// Mitsubishi GX Works2 project: A1-60MR-GX2   PLC: FX3G

PROGRAM MAIN
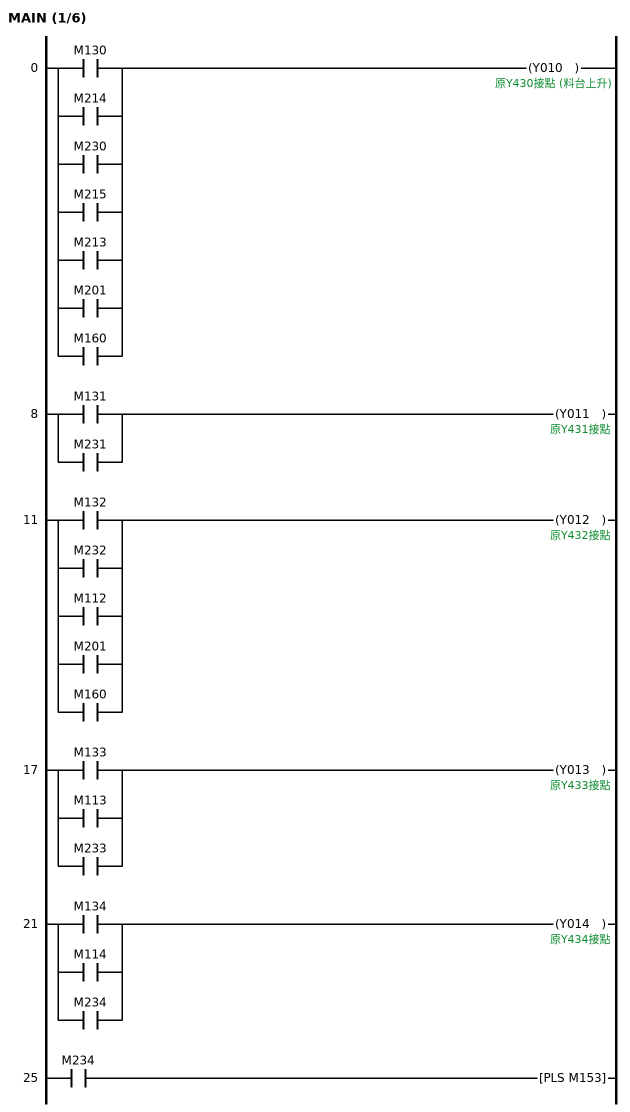
0     LD      M130
      OR      M214
      OR      M230
      OR      M215
      OR      M213
      OR      M201
      OR      M160
      OUT     Y010  ; 原Y430接點 (料台上升)
8     LD      M131
      OR      M231
      OUT     Y011  ; 原Y431接點
11    LD      M132
      OR      M232
      OR      M112
      OR      M201
      OR      M160
      OUT     Y012  ; 原Y432接點
17    LD      M133
      OR      M113
      OR      M233
      OUT     Y013  ; 原Y433接點
21    LD      M134
      OR      M114
      OR      M234
      OUT     Y014  ; 原Y434接點
25    LD      M234
      PLS     M153
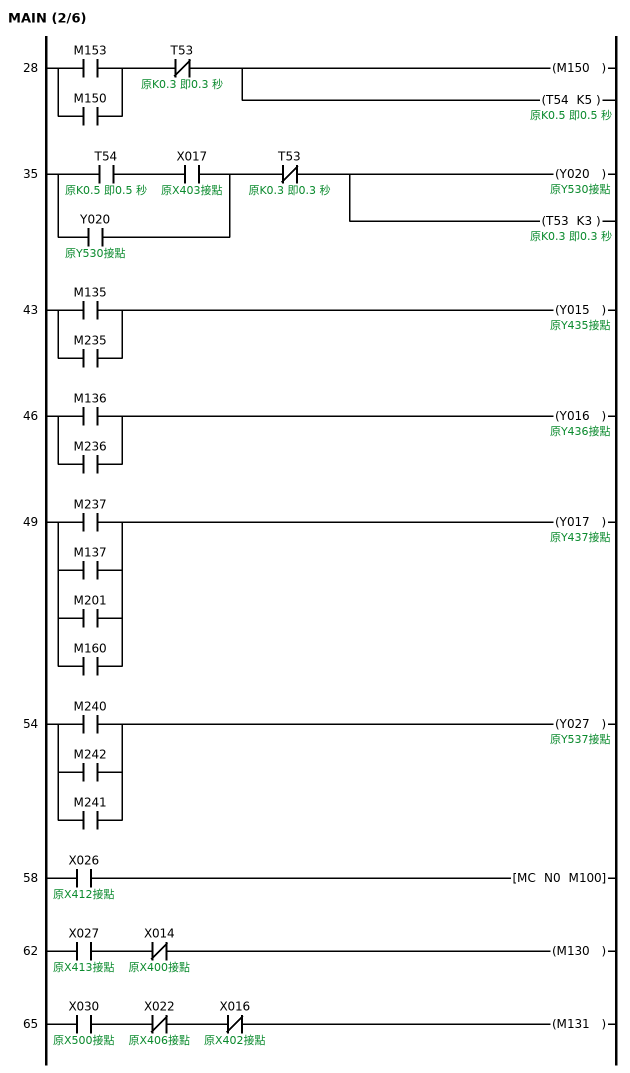
28    LD      M153
      OR      M150
      ANI     T53  ; 原K0.3 即0.3 秒
      OUT     M150
      OUT     T54 K5  ; 原K0.5 即0.5 秒
35    LD      T54  ; 原K0.5 即0.5 秒
      AND     X017  ; 原X403接點
      OR      Y020  ; 原Y530接點
      ANI     T53  ; 原K0.3 即0.3 秒
      OUT     Y020  ; 原Y530接點
      OUT     T53 K3  ; 原K0.3 即0.3 秒
43    LD      M135
      OR      M235
      OUT     Y015  ; 原Y435接點
46    LD      M136
      OR      M236
      OUT     Y016  ; 原Y436接點
49    LD      M237
      OR      M137
      OR      M201
      OR      M160
      OUT     Y017  ; 原Y437接點
54    LD      M240
      OR      M242
      OR      M241
      OUT     Y027  ; 原Y537接點
58    LD      X026  ; 原X412接點
      MC      N0 M100
62    LD      X027  ; 原X413接點
      ANI     X014  ; 原X400接點
      OUT     M130
65    LD      X030  ; 原X500接點
      ANI     X022  ; 原X406接點
      ANI     X016  ; 原X402接點
      OUT     M131
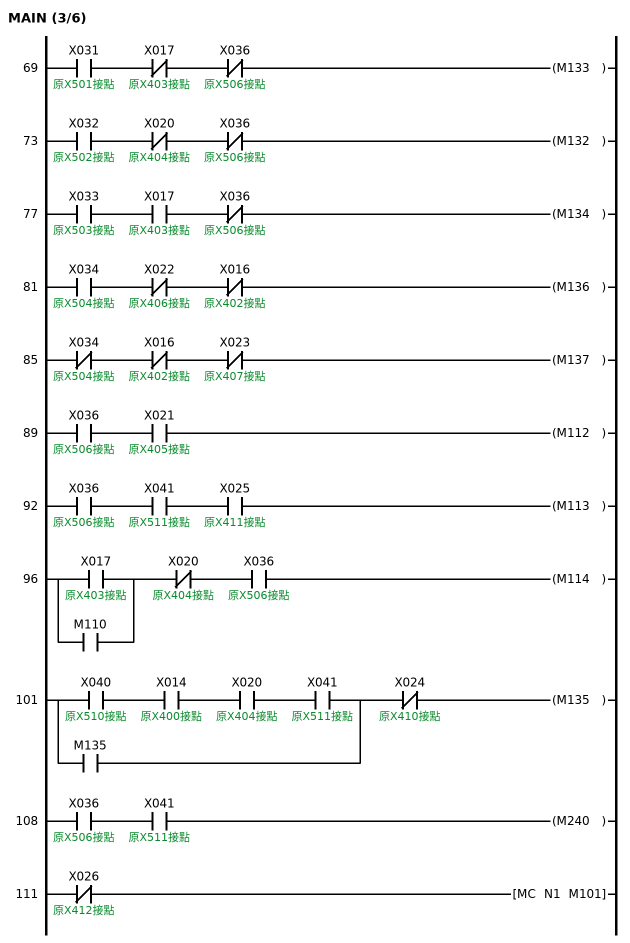
69    LD      X031  ; 原X501接點
      ANI     X017  ; 原X403接點
      ANI     X036  ; 原X506接點
      OUT     M133
73    LD      X032  ; 原X502接點
      ANI     X020  ; 原X404接點
      ANI     X036  ; 原X506接點
      OUT     M132
77    LD      X033  ; 原X503接點
      AND     X017  ; 原X403接點
      ANI     X036  ; 原X506接點
      OUT     M134
81    LD      X034  ; 原X504接點
      ANI     X022  ; 原X406接點
      ANI     X016  ; 原X402接點
      OUT     M136
85    LDI     X034  ; 原X504接點
      ANI     X016  ; 原X402接點
      ANI     X023  ; 原X407接點
      OUT     M137
89    LD      X036  ; 原X506接點
      AND     X021  ; 原X405接點
      OUT     M112
92    LD      X036  ; 原X506接點
      AND     X041  ; 原X511接點
      AND     X025  ; 原X411接點
      OUT     M113
96    LD      X017  ; 原X403接點
      OR      M110
      ANI     X020  ; 原X404接點
      AND     X036  ; 原X506接點
      OUT     M114
101   LD      X040  ; 原X510接點
      AND     X014  ; 原X400接點
      AND     X020  ; 原X404接點
      AND     X041  ; 原X511接點
      OR      M135
      ANI     X024  ; 原X410接點
      OUT     M135
108   LD      X036  ; 原X506接點
      AND     X041  ; 原X511接點
      OUT     M240
111   LDI     X026  ; 原X412接點
      MC      N1 M101
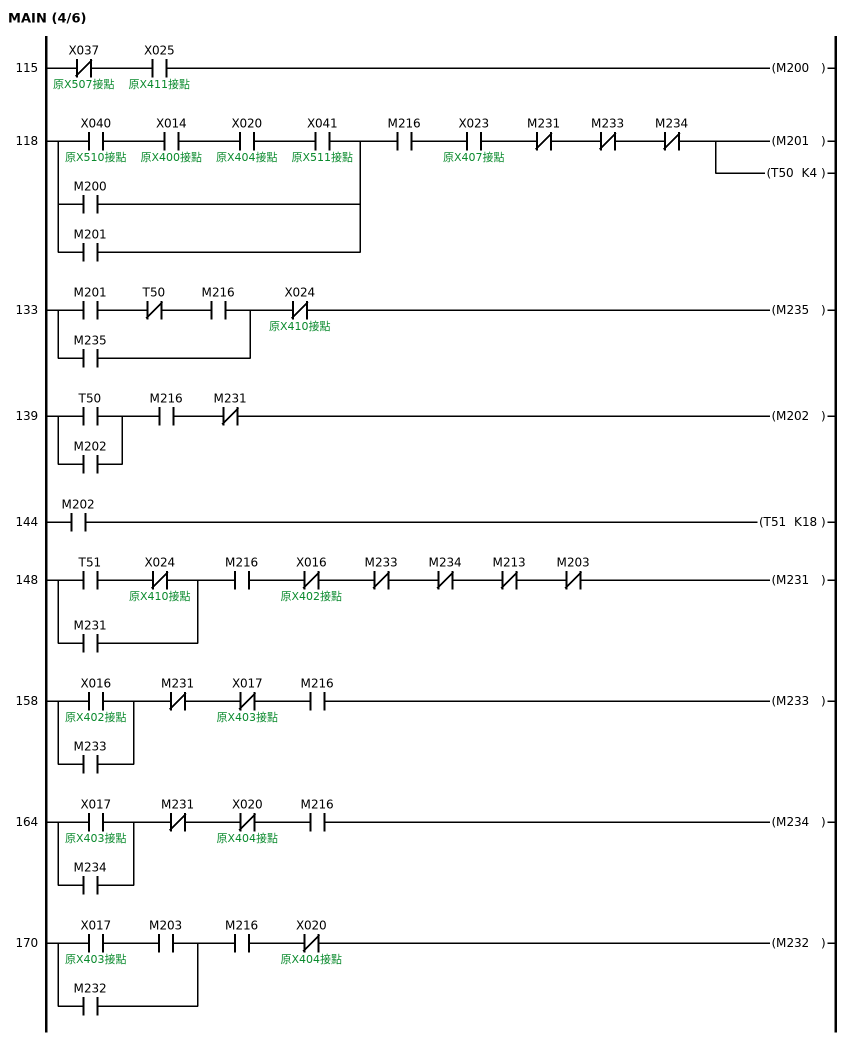
115   LDI     X037  ; 原X507接點
      AND     X025  ; 原X411接點
      OUT     M200
118   LD      X040  ; 原X510接點
      AND     X014  ; 原X400接點
      AND     X020  ; 原X404接點
      AND     X041  ; 原X511接點
      OR      M200
      OR      M201
      AND     M216
      AND     X023  ; 原X407接點
      ANI     M231
      ANI     M233
      ANI     M234
      OUT     M201
      OUT     T50 K4
133   LD      M201
      ANI     T50
      AND     M216
      OR      M235
      ANI     X024  ; 原X410接點
      OUT     M235
139   LD      T50
      OR      M202
      AND     M216
      ANI     M231
      OUT     M202
144   LD      M202
      OUT     T51 K18
148   LD      T51
      ANI     X024  ; 原X410接點
      OR      M231
      AND     M216
      ANI     X016  ; 原X402接點
      ANI     M233
      ANI     M234
      ANI     M213
      ANI     M203
      OUT     M231
158   LD      X016  ; 原X402接點
      OR      M233
      ANI     M231
      ANI     X017  ; 原X403接點
      AND     M216
      OUT     M233
164   LD      X017  ; 原X403接點
      OR      M234
      ANI     M231
      ANI     X020  ; 原X404接點
      AND     M216
      OUT     M234
170   LD      X017  ; 原X403接點
      AND     M203
      OR      M232
      AND     M216
      ANI     X020  ; 原X404接點
      OUT     M232
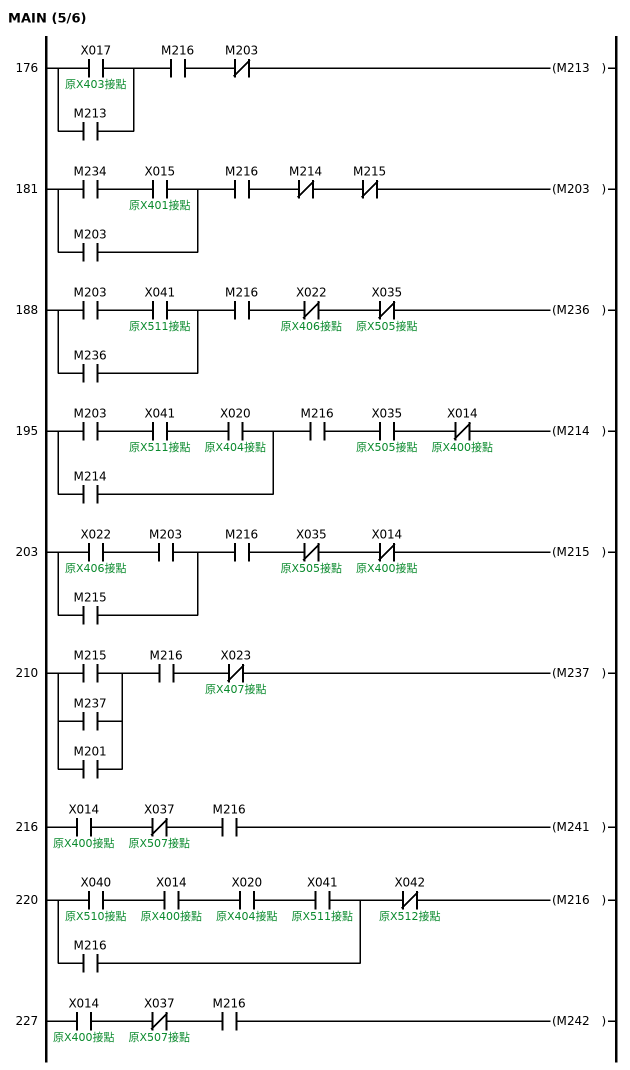
176   LD      X017  ; 原X403接點
      OR      M213
      AND     M216
      ANI     M203
      OUT     M213
181   LD      M234
      AND     X015  ; 原X401接點
      OR      M203
      AND     M216
      ANI     M214
      ANI     M215
      OUT     M203
188   LD      M203
      AND     X041  ; 原X511接點
      OR      M236
      AND     M216
      ANI     X022  ; 原X406接點
      ANI     X035  ; 原X505接點
      OUT     M236
195   LD      M203
      AND     X041  ; 原X511接點
      AND     X020  ; 原X404接點
      OR      M214
      AND     M216
      AND     X035  ; 原X505接點
      ANI     X014  ; 原X400接點
      OUT     M214
203   LD      X022  ; 原X406接點
      AND     M203
      OR      M215
      AND     M216
      ANI     X035  ; 原X505接點
      ANI     X014  ; 原X400接點
      OUT     M215
210   LD      M215
      OR      M237
      OR      M201
      AND     M216
      ANI     X023  ; 原X407接點
      OUT     M237
216   LD      X014  ; 原X400接點
      ANI     X037  ; 原X507接點
      AND     M216
      OUT     M241
220   LD      X040  ; 原X510接點
      AND     X014  ; 原X400接點
      AND     X020  ; 原X404接點
      AND     X041  ; 原X511接點
      OR      M216
      ANI     X042  ; 原X512接點
      OUT     M216
227   LD      X014  ; 原X400接點
      ANI     X037  ; 原X507接點
      AND     M216
      OUT     M242
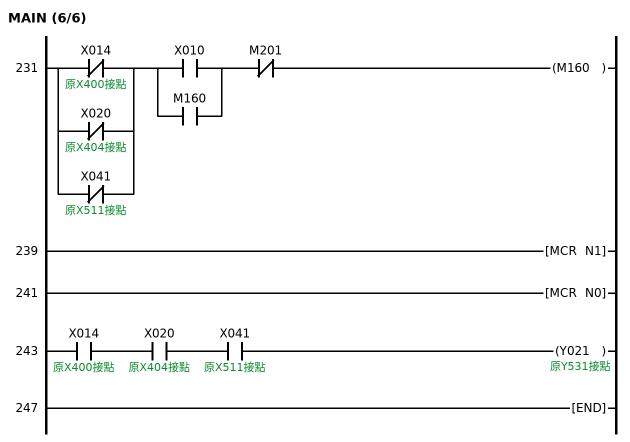
231   LDI     X014  ; 原X400接點
      ORI     X020  ; 原X404接點
      ORI     X041  ; 原X511接點
      LD      X010
      OR      M160
      ANB
      ANI     M201
      OUT     M160
239   MCR     N1
241   MCR     N0
243   LD      X014  ; 原X400接點
      AND     X020  ; 原X404接點
      AND     X041  ; 原X511接點
      OUT     Y021  ; 原Y531接點
247   END
END_PROGRAM

// device comments not shown above
Y022  ; 原Y532接點
Y023  ; 原Y533接點
Y024  ; 原Y534接點
Y025  ; 原Y535接點
Y026  ; 原Y536接點
X043  ; 原X513接點
